// TIA Portal V20 export
// export: Created 2025-12-01T14:57:03.2888936Z, ExportSetting None, DisplayName Totally Integrated Automation Portal, DisplayVersion V20 Update 3, DisplayName TIA Portal Openness, DisplayVersion V20 Update 3, DisplayName TIA Portal Version Control Interface, DisplayVersion V20 Update 3, DisplayName STEP 7 Professional, DisplayVersion V20 Update 3, DisplayName STEP 7 Safety, DisplayVersion V20 Update 2, DisplayName WinCC Basic/Comfort/Advanced, DisplayVersion V20 Update 3, DisplayName WinCC Professional, DisplayVersion V20 Update 3, DisplayName WinCC Unified, DisplayVersion V20 Update 3
FUNCTION "FC666_SIMULTANEIDAD" : Void   // FC666, STL
{ S7_Optimized_Access := 'TRUE' }
// stored: AutoNumber false
   VAR_INPUT
      flanco_registrar : Bool;
   END_VAR
   VAR_TEMP
      Num_Motores_ON : Int;
      N_mesa : Int;
      total_registros : Int;
      offset_primero : Int;
      offset_registros : Int;
      ultimo_guardado : Int;
   END_VAR
BEGIN

NETWORK
TITLE = 
      SET;
      AN    #flanco_registrar;
      JC    salir;



NETWORK
TITLE = SIMULTANEIDAD
// inicialización de datos

      LAR1  P#0.0;


      OPN   "DB666_SIMUL";
      L     DBW [AR1, P#0.0];
      T     #total_registros;
      L     DBW [AR1, P#2.0];
      T     #offset_primero;
      L     DBW [AR1, P#4.0];
      T     #offset_registros;
      L     DBW [AR1, P#6.0];
      T     #ultimo_guardado;


      L     0;
      T     #Num_Motores_ON;
      T     #N_mesa;


      LAR1  P#0.0;




next: OPN   "DB900_Estado_Mesas";
      L     DBB [AR1, P#10.0];
      L     0;
      ==I;
      JC    NoM;

      L     1;
      L     #Num_Motores_ON;
      +I;
      T     #Num_Motores_ON;

NoM:  L     1;
      L     #N_mesa;
      +I;
      T     #N_mesa;
      L     500;
      <=I;
      JC    SIG;

      JU    fin;


SIG:  +AR1  P#16.0;
      JU    next;

//===============================================================


fin:  OPN   "DB666_SIMUL";
      A(;
      L     #ultimo_guardado;
      L     1;
      >=I;
      );
      A(;
      L     #ultimo_guardado;
      L     #total_registros;
      <=I;
      );
      JC    punt;


      L     1;
      T     #ultimo_guardado;

punt: L     #ultimo_guardado;
      L     1;
      -I;
      L     #offset_registros;
      *I;
      L     #offset_primero;
      +I;
      SLD   3;
      LAR1;

      OPN   "DB666_SIMUL";
      L     #Num_Motores_ON;
      T     DBW [AR1, P#0.0];

      L     1;
      L     #ultimo_guardado;
      +I;
      T     #ultimo_guardado;

      LAR1  P#0.0;
      L     #ultimo_guardado;
      T     DBW [AR1, P#6.0];



salir:NOP   0;
END_FUNCTION
